TYPE E_TcMatSimDataAreaType :
(
	NotSpecified := 0,
	Standard,
	InputSrc,
	InputDst,
	OutputSrc,
	OutputDst,
	InternalDa,
	MArea,
	RetainDa
);
END_TYPE

(* stored: Version 1.1.0.1, ProductVersion 3.1.4024.4
   DUT E_TcMatSimDataAreaType: Id {048d1ef5-1995-4917-91cd-dfb17c320419} *)
